// TIA Portal V17 export
// export: Created 2022-07-28T18:02:46.3381407Z, ExportSetting None, DisplayName Totally Integrated Automation Portal, DisplayVersion V17, DisplayName TIA Portal Openness, DisplayVersion V17, DisplayName TIA Portal Teamcenter Gateway, DisplayVersion V17, DisplayName TIA Portal Version Control Interface, DisplayVersion V17, DisplayName TIA Portal Test Suite Advanced, DisplayVersion V17, DisplayName SINAMICS Startdrive Advanced, DisplayVersion V17, DisplayName SINAMICS DCC, DisplayVersion V17, DisplayName SINAMICS Startdrive G130, G150, S120, S150, SINAMICS MV, S210, DisplayVersion V17, DisplayName SINAMICS Startdrive G110M, G120, G120C, G120D, G120P, G115D, DisplayVersion V17, DisplayName STEP 7 Professional, DisplayVersion V17, DisplayName SIMATIC Energy Suite, DisplayVersion V17, DisplayName STEP 7 CFC, DisplayVersion V17, DisplayName STEP 7 Safety, DisplayVersion V17, DisplayName WinCC Advanced / Unified PC, DisplayVersion V17, DisplayName SIMATIC Visualization Architect, DisplayVersion V17
FUNCTION_BLOCK "Lib_FB_Timer_TP_Simple"   // FB13, SCL
{ S7_Optimized_Access := 'TRUE' }
// stored: AutoNumber false, MemoryReserve 100, SetENOAutomatically false
   VAR_INPUT
      IR_CycleTime { ExternalAccessible := 'False'; ExternalVisible := 'False'; ExternalWritable := 'False'} : Real;   // Last cycle time of PLC, s
      IB_StartTimerInput { ExternalAccessible := 'False'; ExternalVisible := 'False'; ExternalWritable := 'False'} : Bool;   // 1 = start timer
      IB_ResetTimer { ExternalAccessible := 'False'; ExternalVisible := 'False'; ExternalWritable := 'False'} : Bool;   // 1 = stop timer. Out = 0
      IR_SpTime { ExternalAccessible := 'False'; ExternalVisible := 'False'; ExternalWritable := 'False'} : Real;   // Setpoint time for timer, s
   END_VAR
   VAR_OUTPUT
      QB_TimerOut { ExternalAccessible := 'False'; ExternalVisible := 'False'; ExternalWritable := 'False'} : Bool;   // 1 = timer done
   END_VAR
   VAR
      sStartTimer { ExternalAccessible := 'False'; ExternalVisible := 'False'; ExternalWritable := 'False'} : Bool;   // To out signal
      sOldIn : Bool;   // Old value of timer input
      sR_Cv_ToDone { ExternalWritable := 'False'} : Real;   // Час до завешення відліку
   END_VAR
   VAR_TEMP
      tmp_QB_TimerOut : Bool;
      tNotDone : Bool;
   END_VAR
BEGIN
   //-------------------------------------
   IF  NOT #sStartTimer
   THEN
       #sR_Cv_ToDone := #IR_SpTime;
   END_IF;
   //-------------------------------------
   //-------------------------------------
   IF #IB_ResetTimer
   THEN
       #sR_Cv_ToDone := -1.0;
   END_IF;
   //-------------------------------------

   #tNotDone := (#sR_Cv_ToDone > 0);

   #sStartTimer := ((#IB_StartTimerInput AND NOT #sOldIn)
   OR (#sStartTimer AND #tNotDone))
   AND NOT #IB_ResetTimer;

   #sOldIn := #IB_StartTimerInput;

   //-------------------------------------
   IF #sStartTimer AND #tNotDone THEN
       //коли була зміна завдання
       IF #sR_Cv_ToDone >= #IR_SpTime
       THEN
           #sR_Cv_ToDone := #IR_SpTime;
       END_IF;
       //--------------------------------------------
       #sR_Cv_ToDone := #sR_Cv_ToDone - #IR_CycleTime;
   END_IF;
   //--------------------------------------------
   #tmp_QB_TimerOut := #sR_Cv_ToDone > 0
   AND #sStartTimer;
   #QB_TimerOut := #tmp_QB_TimerOut;
END_FUNCTION_BLOCK
